VAR_GLOBAL
	stEL6001InIMU1 AT %I*	: EL6inData22B;		//**To EL6021 Inputs**
	stEL6001OutIMU1 AT %Q*	: EL6outData22B;	//**To EL6021 Outputs**
	
	stEL6001InIMU2 AT %I*	: EL6inData22B;		//**To EL6021 Inputs**
	stEL6001OutIMU2 AT %Q*	: EL6outData22B;	//**To EL6021 Outputs**
END_VAR

(* stored: Version 1.1.0.1, ProductVersion 3.1.4024.12
   GVL AccelerationSensor: Id {3e4349e6-a99a-4aa8-b94a-96e30307ccae} *)
